TYPE FsT_ErrCode : LINT; END_TYPE

(* stored: Version 1.1.0.1, ProductVersion 3.1.4024.4
   DUT FsT_ErrCode: Id {2480f718-c38e-4752-b484-05959eedf60a} *)
